PROGRAM MAPPING_in
VAR
  bFirstCycle           : BOOL := TRUE;

  AxisState             : U_AXIS_STATE;
  AxisInfo              : U_AXIS_INFO;
  AxisParameterRd       : U_AXIS_NC_PARAMETER_RD;

  CamState              : U_CAM_STATE;
  CamInfo               : U_CAM_INFO;

  TriggerState          : U_TRIGGER_STATE;

  TouchState            : U_TOUCH_PROBE_STATE;

  FlyState              : U_FLY_STATE;


  szAxisPara,
  szAxisInfo,
  szAxisState           : ARRAY[1..2] OF UDINT;

  szCamInfo,
  szCamData,
  szCamState            : ARRAY[1..2] OF UDINT;

  szStateTouchProbe,
  szStateTrigger	      :  ARRAY[1..2] OF UDINT;
END_VAR


IF (bFirstCycle)
THEN
  bFirstCycle         := FALSE;
  
  szAxisState[1]      := SIZEOF(AxisState);
  szAxisState[2]      := SIZEOF(GVL_AXIS.State);
  
  szAxisInfo [1]      := SIZEOF(AxisInfo);
  szAxisInfo [2]      := SIZEOF(GVL_AXIS.Info);
  
  szAxisPara [1]      := SIZEOF(AxisParameterRd);
  szAxisPara [2]      := SIZEOF(GVL_AXIS.NcParameterRd);
END_IF

  memcpy(ADR(GVL_AXIS.State),             ADR(AxisState),              SIZEOF(AxisState));
  memcpy(ADR(GVL_AXIS.Info),              ADR(AxisInfo),               SIZEOF(AxisInfo));
  memcpy(ADR(GVL_AXIS.NcParameterRd),     ADR(AxisParameterRd),        SIZEOF(AxisParameterRd));

  memcpy(ADR(GVL_CAM.State),              ADR(CamState),               SIZEOF(CamState));
  memcpy(ADR(GVL_CAM.Info),               ADR(CamInfo),                SIZEOF(CamInfo));

  memcpy(ADR(GVL_FUNCTIONS.StateTrigger),    ADR(TriggerState),        SIZEOF(TriggerState));
  memcpy(ADR(GVL_FUNCTIONS.StateTouchProbe), ADR(TouchState),          SIZEOF(TouchState));

  memcpy(ADR(GVL_FLYING_SAW.State),       ADR(FlyState),               SIZEOF(FlyState));

END_PROGRAM

(* stored: Version 1.1.0.1
   POU MAPPING_in: Id {9c1c55cc-539c-4e24-8b74-c3ec7fa50c1e}, SpecialFunc None *)
